FUNCTION_BLOCK Vertical_process
VAR_INPUT
	activate: BOOL;
END_VAR
VAR_OUTPUT
	done: BOOL;
END_VAR
VAR
	TOF_1: TOF;
	R_TRIG_0: R_TRIG;
	F_TRIG_0: F_TRIG;
	TOF_0: TOF;
END_VAR
VAR // added by the converter: edge detectors and wires of the graphical bodies
    _w1 : BOOL;
END_VAR

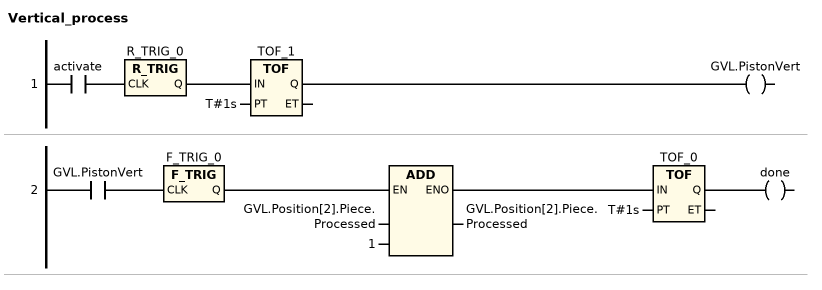
// NETWORK 1
R_TRIG_0(CLK := activate); // R_TRIG
TOF_1(IN := R_TRIG_0.Q, PT := T#1s); // TOF
GVL.PistonVert := TOF_1.Q;

// NETWORK 2
F_TRIG_0(CLK := GVL.PistonVert); // F_TRIG
_w1 := F_TRIG_0.Q;
IF _w1 THEN GVL.Position[2].Piece.Processed := GVL.Position[2].Piece.Processed + 1; END_IF
TOF_0(IN := _w1, PT := T#1s); // TOF
done := TOF_0.Q;

END_FUNCTION_BLOCK

(* stored: Version 1.1.0.1, ProductVersion 3.1.4024.12
   POU Vertical_process: Id {01bc5ec2-9a83-45f3-b0d9-241c51c6ca34}, SpecialFunc None *)
